(* IEC 61131-3 sources: stc/tests/corpus/agents4plc, 4 files *)

(* ---- st_file_20251118180902.st ---- *)
FUNCTION_BLOCK MultiPumpCtrl
VAR_INPUT
    mode : BOOL;
    start : BOOL;
    stop : BOOL;
    priorities : ARRAY[1..5] OF INT;
    selections : ARRAY[1..5] OF BOOL;
END_VAR
VAR_OUTPUT
    RunComds : ARRAY[1..5] OF BOOL;
END_VAR
VAR
    i : INT;
    j : INT;
    maxPriority : INT;
    maxIndex : INT;
    runCount : INT;
    usedInAuto : ARRAY[1..5] OF BOOL;
END_VAR

(* Stop signal has highest priority *)
IF stop THEN
    FOR i := 1 TO 5 DO
        RunComds[i] := FALSE;
    END_FOR;
ELSE
    (* Mode selection logic *)
    IF NOT mode THEN (* Manual mode *)
        IF start THEN
            FOR i := 1 TO 5 DO
                RunComds[i] := selections[i];
            END_FOR;
        END_IF;
    ELSE (* Automatic mode *)
        IF start THEN
            (* Initialize usedInAuto array *)
            FOR i := 1 TO 5 DO
                usedInAuto[i] := FALSE;
            END_FOR;

            runCount := 0;

            (* Find 3 highest priority pumps *)
            WHILE runCount < 3 DO
                maxPriority := -32768; (* Minimum INT value *)
                maxIndex := 0;

                (* Find highest priority pump not already used *)
                FOR i := 1 TO 5 DO
                    IF (priorities[i] > maxPriority) AND NOT usedInAuto[i] THEN
                        maxPriority := priorities[i];
                        maxIndex := i;
                    END_IF;
                END_FOR;

                (* Mark pump as used and set run command *)
                IF maxIndex > 0 THEN
                    usedInAuto[maxIndex] := TRUE;
                    RunComds[maxIndex] := TRUE;
                    runCount := runCount + 1;
                END_IF;
            END_WHILE;

            (* Set remaining pumps to FALSE *)
            FOR i := 1 TO 5 DO
                IF NOT usedInAuto[i] THEN
                    RunComds[i] := FALSE;
                END_IF;
            END_FOR;
        END_IF;
    END_IF;
END_IF;
END_FUNCTION_BLOCK

(* ---- st_file_20251118180959.st ---- *)
FUNCTION_BLOCK MultiPumpCtrl
VAR_INPUT
    mode : BOOL;
    start : BOOL;
    stop : BOOL;
    priorities : ARRAY[1..5] OF INT;
    selections : ARRAY[1..5] OF BOOL;
END_VAR
VAR_OUTPUT
    RunComds : ARRAY[1..5] OF BOOL;
END_VAR
VAR
    i : INT;
    j : INT;
    maxPriority : INT;
    maxIndex : INT;
    runCount : INT;
    usedInAuto : ARRAY[1..5] OF BOOL;
END_VAR
(* Always clear commands first *)
FOR i := 1 TO 5 DO
    RunComds[i] := FALSE;
END_FOR;

(* Stop signal has absolute priority *)
IF NOT stop THEN
    (* Mode selection logic *)
    IF NOT mode THEN (* Manual mode *)
        IF start THEN
            FOR i := 1 TO 5 DO
                RunComds[i] := selections[i];
            END_FOR;
        END_IF;
    ELSE (* Automatic mode *)
        IF start THEN
            (* Initialize usedInAuto array *)
            FOR i := 1 TO 5 DO
                usedInAuto[i] := FALSE;
            END_FOR;

            runCount := 0;

            (* Find 3 highest priority pumps *)
            WHILE runCount < 3 DO
                maxPriority := -32768; (* Minimum INT value *)
                maxIndex := 0;

                (* Find highest priority pump not already used *)
                FOR i := 1 TO 5 DO
                    IF (priorities[i] > maxPriority) AND NOT usedInAuto[i] THEN
                        maxPriority := priorities[i];
                        maxIndex := i;
                    END_IF;
                END_FOR;

                (* Mark pump as used and set run command *)
                IF maxIndex > 0 THEN
                    usedInAuto[maxIndex] := TRUE;
                    RunComds[maxIndex] := TRUE;
                    runCount := runCount + 1;
                END_IF;
            END_WHILE;
        END_IF;
    END_IF;
END_IF;

(* Stop signal has highest priority *)
    (* Mode selection logic *)
    IF NOT mode THEN (* Manual mode *)
        IF start THEN
            FOR i := 1 TO 5 DO
                RunComds[i] := selections[i];
            END_FOR;
        END_IF;
    ELSE (* Automatic mode *)
        IF start THEN
            (* Initialize usedInAuto array *)
            FOR i := 1 TO 5 DO
                usedInAuto[i] := FALSE;
            END_FOR;

            runCount := 0;

            (* Find 3 highest priority pumps *)
            WHILE runCount < 3 DO
                maxPriority := -32768; (* Minimum INT value *)
                maxIndex := 0;

                (* Find highest priority pump not already used *)
                FOR i := 1 TO 5 DO
                    IF (priorities[i] > maxPriority) AND NOT usedInAuto[i] THEN
                        maxPriority := priorities[i];
                        maxIndex := i;
                    END_IF;
                END_FOR;

                (* Mark pump as used and set run command *)
                IF maxIndex > 0 THEN
                    usedInAuto[maxIndex] := TRUE;
                    RunComds[maxIndex] := TRUE;
                    runCount := runCount + 1;
                END_IF;
            END_WHILE;

            (* Set remaining pumps to FALSE *)
            FOR i := 1 TO 5 DO
                IF NOT usedInAuto[i] THEN
                    RunComds[i] := FALSE;
                END_IF;
            END_FOR;
        END_IF;
    END_IF;
END_FUNCTION_BLOCK

(* ---- st_file_20251118181045.st ---- *)
FUNCTION_BLOCK MultiPumpCtrl
VAR_INPUT
    mode : BOOL;
    start : BOOL;
    stop : BOOL;
    priorities : ARRAY[1..5] OF INT;
    selections : ARRAY[1..5] OF BOOL;
END_VAR
VAR_OUTPUT
    RunComds : ARRAY[1..5] OF BOOL;
END_VAR
VAR
    i : INT;
    j : INT;
    maxPriority : INT;
    maxIndex : INT;
    runCount : INT;
    usedInAuto : ARRAY[1..5] OF BOOL;
END_VAR
(* Always clear commands first *)
FOR i := 1 TO 5 DO
    RunComds[i] := FALSE;
END_FOR;

(* Stop signal has absolute priority *)
IF stop THEN
    FOR i := 1 TO 5 DO
        RunComds[i] := FALSE;
    END_FOR;
ELSE
    (* Mode selection logic *)
    IF NOT mode THEN (* Manual mode *)
        IF start THEN
            FOR i := 1 TO 5 DO
                RunComds[i] := selections[i];
            END_FOR;
        END_IF;
    ELSE (* Automatic mode *)
        IF start THEN
            (* Initialize usedInAuto array *)
            FOR i := 1 TO 5 DO
                usedInAuto[i] := FALSE;
            END_FOR;

            runCount := 0;

            (* Find 3 highest priority pumps *)
            WHILE runCount < 3 DO
                maxPriority := -32768; (* Minimum INT value *)
                maxIndex := 0;

                (* Find highest priority pump not already used *)
                FOR i := 1 TO 5 DO
                    IF (priorities[i] > maxPriority) AND NOT usedInAuto[i] THEN
                        maxPriority := priorities[i];
                        maxIndex := i;
                    END_IF;
                END_FOR;

                (* Mark pump as used and set run command *)
                IF maxIndex > 0 THEN
                    usedInAuto[maxIndex] := TRUE;
                    RunComds[maxIndex] := TRUE;
                    runCount := runCount + 1;
                END_IF;
            END_WHILE;
        END_IF;
    END_IF;
END_IF;

(* Stop signal has highest priority *)
    (* Mode selection logic *)
    IF NOT mode THEN (* Manual mode *)
        IF start THEN
            FOR i := 1 TO 5 DO
                RunComds[i] := selections[i];
            END_FOR;
        END_IF;
    ELSE (* Automatic mode *)
        IF start THEN
            (* Initialize usedInAuto array *)
            FOR i := 1 TO 5 DO
                usedInAuto[i] := FALSE;
            END_FOR;

            runCount := 0;

            (* Find 3 highest priority pumps *)
            WHILE runCount < 3 DO
                maxPriority := -32768; (* Minimum INT value *)
                maxIndex := 0;

                (* Find highest priority pump not already used *)
                FOR i := 1 TO 5 DO
                    IF (priorities[i] > maxPriority) AND NOT usedInAuto[i] THEN
                        maxPriority := priorities[i];
                        maxIndex := i;
                    END_IF;
                END_FOR;

                (* Mark pump as used and set run command *)
                IF maxIndex > 0 THEN
                    usedInAuto[maxIndex] := TRUE;
                    RunComds[maxIndex] := TRUE;
                    runCount := runCount + 1;
                END_IF;
            END_WHILE;

            (* Set remaining pumps to FALSE *)
            FOR i := 1 TO 5 DO
                IF NOT usedInAuto[i] THEN
                    RunComds[i] := FALSE;
                END_IF;
            END_FOR;
        END_IF;
    END_IF;
END_FUNCTION_BLOCK

(* ---- st_file_20251120154545.st ---- *)
FUNCTION_BLOCK StackMin
VAR_INPUT
    push : BOOL;
    pop : BOOL;
    reset : BOOL;
END_VAR
VAR_OUTPUT
    error : BOOL;
    status : WORD;
END_VAR
VAR_IN_OUT
    item : INT;
    stack : ARRAY[0..3] OF INT;
END_VAR
VAR
    top : INT := -1;
    min_index : INT;
    i : INT;
    temp_min : INT;
END_VAR

(* Reset has highest priority *)
IF reset THEN
    top := -1;
    error := FALSE;
    status := 16#0000;
(* Push operation *)
ELSIF push THEN
    IF top = 3 THEN
        error := TRUE;
        status := 16#8A04;
    ELSE
        top := top + 1;
        stack[top] := item;
        error := FALSE;
        status := 16#0000;
    END_IF;
(* Pop operation *)
ELSIF pop THEN
    IF top = -1 THEN
        error := TRUE;
        status := 16#8A05;
    ELSE
        (* Find minimum value and its index *)
        min_index := 0;
        temp_min := stack[0];
        FOR i := 1 TO top DO
            IF stack[i] < temp_min THEN
                temp_min := stack[i];
                min_index := i;
            END_IF;
        END_FOR;

        (* Store min value in output *)
        item := temp_min;

        (* Shift elements down *)
        FOR i := min_index TO top - 1 DO
            stack[i] := stack[i + 1];
        END_FOR;

        (* Decrement top *)
        top := top - 1;
        error := FALSE;
        status := 16#0000;
    END_IF;
(* No operation - clear error state *)
ELSE
    error := FALSE;
    status := 16#0000;
END_IF;
END_FUNCTION_BLOCK
